Fanuc TP program (LS listing): _set_rack_slot.ls

/PROG  _SET_RACK_SLOT
/ATTR
OWNER		= MNEDITOR;
COMMENT		= "";
PROG_SIZE	= 6875;
CREATE		= DATE 26-07-16  TIME 09:15:24;
MODIFIED	= DATE 26-07-17  TIME 00:46:46;
FILE_NAME	= ;
VERSION		= 0;
LINE_COUNT	= 333;
MEMORY_SIZE	= 7591;
PROTECT		= READ_WRITE;
TCD:  STACK_SIZE	= 0,
      TASK_PRIORITY	= 50,
      TIME_SLICE	= 0,
      BUSY_LAMP_OFF	= 0,
      ABORT_REQUEST	= 0,
      PAUSE_REQUEST	= 0;
DEFAULT_GROUP	= 1,*,*,*,*;
CONTROL_CODE	= 00000000 00000000;
LOCAL_REGISTERS	= 0,0,0;
/APPL

AUTO_SINGULARITY_HEADER;
  ENABLE_SINGULARITY_AVOIDANCE   : TRUE;
/MN
   1:  !*******SET RACK PKPL SLOT******* ;
   2:  LBL[100] ;
   3:  F[21:OFF:Rack Slot-Set]=(OFF) ;
   4:  !**Jump for Rack to PKPL at ;
   5:  SELECT R[20:*RackNum]=1,JMP LBL[210] ;
   6:         =2,JMP LBL[220] ;
   7:         =3,JMP LBL[230] ;
   8:         =4,JMP LBL[240] ;
   9:         =5,JMP LBL[250] ;
  10:         =6,JMP LBL[260] ;
  11:  JMP LBL[700] ;
  12:   ;
  13:  !***Rack-1 (Door)**************** ;
  14:  LBL[210] ;
  15:  !Jump for Column ;
  16:  SELECT R[25:*Slot-Colmn]=1,JMP LBL[211] ;
  17:         =2,JMP LBL[212] ;
  18:         =3,JMP LBL[213] ;
  19:         =4,JMP LBL[214] ;
  20:  JMP LBL[700] ;
  21:   ;
  22:  !**Column 1-Chk Row  ;
  23:  LBL[211] ;
  24:  IF (R[26:*Slot-Row]<1 OR R[26:*Slot-Row]>7),JMP LBL[700] ;
  25:  !Set Origin PR ;
  26:  R[27:*RackOrig-PR]=161    ;
  27:  !Set Appr PR/Transit Angle ;
  28:  R[28:*RackAppr-PR]=131    ;
  29:  R[24:*TransitAngle]=(-155)    ;
  30:  JMP LBL[300] ;
  31:   ;
  32:  !**Column 2-Chk Row  ;
  33:  LBL[212] ;
  34:  IF (R[26:*Slot-Row]<>1 AND R[26:*Slot-Row]<>2),JMP LBL[700] ;
  35:  !Set Origin PR ;
  36:  R[27:*RackOrig-PR]=162    ;
  37:  !Set Appr PR/Transit Angle ;
  38:  R[28:*RackAppr-PR]=131    ;
  39:  R[24:*TransitAngle]=(-155)    ;
  40:  JMP LBL[300] ;
  41:   ;
  42:  !**Column 3-Chk Row  ;
  43:  LBL[213] ;
  44:  IF (R[26:*Slot-Row]<>1 AND R[26:*Slot-Row]<>2),JMP LBL[700] ;
  45:  !Set Origin PR ;
  46:  R[27:*RackOrig-PR]=163    ;
  47:  !Set Appr PR/Transit Angle ;
  48:  R[28:*RackAppr-PR]=132    ;
  49:  R[24:*TransitAngle]=155    ;
  50:  JMP LBL[300] ;
  51:   ;
  52:  !**Column 4-Chk Row  ;
  53:  LBL[214] ;
  54:  IF (R[26:*Slot-Row]<1 OR R[26:*Slot-Row]>6),JMP LBL[700] ;
  55:  !Set Origin PR ;
  56:  R[27:*RackOrig-PR]=164    ;
  57:  !Set Appr PR/Transit Angle ;
  58:  R[28:*RackAppr-PR]=132    ;
  59:  R[24:*TransitAngle]=155    ;
  60:  JMP LBL[300] ;
  61:   ;
  62:   ;
  63:  !***Rack-2 (Full)**************** ;
  64:  LBL[220] ;
  65:  !Jump for Column ;
  66:  SELECT R[25:*Slot-Colmn]=1,JMP LBL[221] ;
  67:         =2,JMP LBL[222] ;
  68:         =3,JMP LBL[223] ;
  69:         =4,JMP LBL[224] ;
  70:  JMP LBL[700] ;
  71:   ;
  72:  !**Column 1-Chk Row  ;
  73:  LBL[221] ;
  74:  IF (R[26:*Slot-Row]<1 OR R[26:*Slot-Row]>7),JMP LBL[700] ;
  75:  !Set Origin PR ;
  76:  R[27:*RackOrig-PR]=166    ;
  77:  !Set Appr PR/Transit Angle ;
  78:  R[28:*RackAppr-PR]=133    ;
  79:  R[24:*TransitAngle]=(-95)    ;
  80:  JMP LBL[300] ;
  81:   ;
  82:  !**Column 2-Chk Row  ;
  83:  LBL[222] ;
  84:  IF (R[26:*Slot-Row]<1 OR R[26:*Slot-Row]>7),JMP LBL[700] ;
  85:  !Set Origin PR ;
  86:  R[27:*RackOrig-PR]=167    ;
  87:  !Set Appr PR/Transit Angle ;
  88:  R[28:*RackAppr-PR]=133    ;
  89:  R[24:*TransitAngle]=(-95)    ;
  90:  JMP LBL[300] ;
  91:   ;
  92:  !**Column 3-Chk Row  ;
  93:  LBL[223] ;
  94:  IF (R[26:*Slot-Row]<1 OR R[26:*Slot-Row]>7),JMP LBL[700] ;
  95:  !Set Origin PR ;
  96:  R[27:*RackOrig-PR]=168    ;
  97:  !Set Appr PR/Transit Angle ;
  98:  R[28:*RackAppr-PR]=134    ;
  99:  R[24:*TransitAngle]=(-145)    ;
 100:  JMP LBL[300] ;
 101:   ;
 102:  !**Column 4-Chk Row  ;
 103:  LBL[224] ;
 104:  IF (R[26:*Slot-Row]<1 OR R[26:*Slot-Row]>6),JMP LBL[700] ;
 105:  !Set Origin PR ;
 106:  R[27:*RackOrig-PR]=169    ;
 107:  !Set Appr PR/Transit Angle ;
 108:  R[28:*RackAppr-PR]=134    ;
 109:  R[24:*TransitAngle]=(-145)    ;
 110:  JMP LBL[300] ;
 111:   ;
 112:   ;
 113:  !***Rack-3 (Convs)*************** ;
 114:  LBL[230] ;
 115:  !Jump for Column ;
 116:  SELECT R[25:*Slot-Colmn]=1,JMP LBL[231] ;
 117:         =2,JMP LBL[232] ;
 118:         =3,JMP LBL[233] ;
 119:         =4,JMP LBL[234] ;
 120:  JMP LBL[700] ;
 121:   ;
 122:  !**Column 1-Chk Row  ;
 123:  LBL[231] ;
 124:  IF (R[26:*Slot-Row]<1 OR R[26:*Slot-Row]>4),JMP LBL[700] ;
 125:  !Set Origin PR ;
 126:  R[27:*RackOrig-PR]=171    ;
 127:  !Set Appr PR/Transit Angle ;
 128:  R[28:*RackAppr-PR]=135    ;
 129:  R[24:*TransitAngle]=(-35)    ;
 130:  JMP LBL[300] ;
 131:   ;
 132:  !**Column 2-Chk Row  ;
 133:  LBL[232] ;
 134:  IF (R[26:*Slot-Row]<1 OR R[26:*Slot-Row]>4),JMP LBL[700] ;
 135:  !Set Origin PR ;
 136:  R[27:*RackOrig-PR]=172    ;
 137:  !Set Appr PR/Transit Angle ;
 138:  R[28:*RackAppr-PR]=135    ;
 139:  R[24:*TransitAngle]=(-35)    ;
 140:  JMP LBL[300] ;
 141:   ;
 142:  !**Column 3-Chk Row  ;
 143:  LBL[233] ;
 144:  IF (R[26:*Slot-Row]<1 OR R[26:*Slot-Row]>4),JMP LBL[700] ;
 145:  !Set Origin PR ;
 146:  R[27:*RackOrig-PR]=173    ;
 147:  !Set Appr PR/Transit Angle ;
 148:  R[28:*RackAppr-PR]=136    ;
 149:  R[24:*TransitAngle]=(-85)    ;
 150:  JMP LBL[300] ;
 151:   ;
 152:  !**Column 4-Chk Row  ;
 153:  LBL[234] ;
 154:  IF (R[26:*Slot-Row]<1 OR R[26:*Slot-Row]>4),JMP LBL[700] ;
 155:  !Set Origin PR ;
 156:  R[27:*RackOrig-PR]=174    ;
 157:  !Set Appr PR/Transit Angle ;
 158:  R[28:*RackAppr-PR]=136    ;
 159:  R[24:*TransitAngle]=(-85)    ;
 160:  JMP LBL[300] ;
 161:   ;
 162:   ;
 163:  !***Rack-4 (Hopper)************** ;
 164:  LBL[240] ;
 165:  !Jump for Column ;
 166:  SELECT R[25:*Slot-Colmn]=1,JMP LBL[241] ;
 167:         =2,JMP LBL[242] ;
 168:         =3,JMP LBL[243] ;
 169:         =4,JMP LBL[244] ;
 170:  JMP LBL[700] ;
 171:   ;
 172:  !**Column 1-Chk Row  ;
 173:  LBL[241] ;
 174:  IF (R[26:*Slot-Row]<>1 AND R[26:*Slot-Row]<>6 AND R[26:*Slot-Row]<>7),JMP LBL[700] ;
 175:  !Set Origin PR ;
 176:  R[27:*RackOrig-PR]=176    ;
 177:  !Set Appr PR/Transit Angle ;
 178:  R[28:*RackAppr-PR]=137    ;
 179:  R[24:*TransitAngle]=25    ;
 180:  JMP LBL[300] ;
 181:   ;
 182:  !**Column 2-Chk Row  ;
 183:  LBL[242] ;
 184:  IF (R[26:*Slot-Row]<>1 AND R[26:*Slot-Row]<>6 AND R[26:*Slot-Row]<>7),JMP LBL[700] ;
 185:  !Set Origin PR ;
 186:  R[27:*RackOrig-PR]=177    ;
 187:  !Set Appr PR/Transit Angle ;
 188:  R[28:*RackAppr-PR]=137    ;
 189:  R[24:*TransitAngle]=25    ;
 190:  JMP LBL[300] ;
 191:   ;
 192:  !**Column 3-Chk Row  ;
 193:  LBL[243] ;
 194:  IF (R[26:*Slot-Row]<>1 AND R[26:*Slot-Row]<>6 AND R[26:*Slot-Row]<>7),JMP LBL[700] ;
 195:  !Set Origin PR ;
 196:  R[27:*RackOrig-PR]=178    ;
 197:  !Set Appr PR/Transit Angle ;
 198:  R[28:*RackAppr-PR]=138    ;
 199:  R[24:*TransitAngle]=(-25)    ;
 200:  JMP LBL[300] ;
 201:   ;
 202:  !**Column 4-Chk Row  ;
 203:  LBL[244] ;
 204:  IF (R[26:*Slot-Row]<1 OR R[26:*Slot-Row]>7),JMP LBL[700] ;
 205:  !Set Origin PR ;
 206:  R[27:*RackOrig-PR]=179    ;
 207:  !Set Appr PR/Transit Angle ;
 208:  R[28:*RackAppr-PR]=138    ;
 209:  R[24:*TransitAngle]=(-25)    ;
 210:  JMP LBL[300] ;
 211:   ;
 212:   ;
 213:  !***Rack-5 (Full)**************** ;
 214:  LBL[250] ;
 215:  !Jump for Column ;
 216:  SELECT R[25:*Slot-Colmn]=1,JMP LBL[251] ;
 217:         =2,JMP LBL[252] ;
 218:         =3,JMP LBL[253] ;
 219:         =4,JMP LBL[254] ;
 220:  JMP LBL[700] ;
 221:   ;
 222:  !**Column 1-Chk Row  ;
 223:  LBL[251] ;
 224:  IF (R[26:*Slot-Row]<1 OR R[26:*Slot-Row]>7),JMP LBL[700] ;
 225:  !Set Origin PR ;
 226:  R[27:*RackOrig-PR]=181    ;
 227:  !Set Appr PR/Transit Angle ;
 228:  R[28:*RackAppr-PR]=139    ;
 229:  R[24:*TransitAngle]=85    ;
 230:  JMP LBL[300] ;
 231:   ;
 232:  !**Column 2-Chk Row  ;
 233:  LBL[252] ;
 234:  IF (R[26:*Slot-Row]<1 OR R[26:*Slot-Row]>7),JMP LBL[700] ;
 235:  !Set Origin PR ;
 236:  R[27:*RackOrig-PR]=182    ;
 237:  !Set Appr PR/Transit Angle ;
 238:  R[28:*RackAppr-PR]=139    ;
 239:  R[24:*TransitAngle]=85    ;
 240:  JMP LBL[300] ;
 241:   ;
 242:  !**Column 3-Chk Row  ;
 243:  LBL[253] ;
 244:  IF (R[26:*Slot-Row]<1 OR R[26:*Slot-Row]>7),JMP LBL[700] ;
 245:  !Set Origin PR ;
 246:  R[27:*RackOrig-PR]=183    ;
 247:  !Set Appr PR/Transit Angle ;
 248:  R[28:*RackAppr-PR]=140    ;
 249:  R[24:*TransitAngle]=35    ;
 250:  JMP LBL[300] ;
 251:   ;
 252:  !**Column 4-Chk Row  ;
 253:  LBL[254] ;
 254:  IF (R[26:*Slot-Row]<1 OR R[26:*Slot-Row]>7),JMP LBL[700] ;
 255:  !Set Origin PR ;
 256:  R[27:*RackOrig-PR]=184    ;
 257:  !Set Appr PR/Transit Angle ;
 258:  R[28:*RackAppr-PR]=140    ;
 259:  R[24:*TransitAngle]=35    ;
 260:  JMP LBL[300] ;
 261:   ;
 262:   ;
 263:  !***Rack-6 (Full)**************** ;
 264:  LBL[260] ;
 265:  !Jump for Column ;
 266:  SELECT R[25:*Slot-Colmn]=1,JMP LBL[261] ;
 267:         =2,JMP LBL[262] ;
 268:         =3,JMP LBL[263] ;
 269:         =4,JMP LBL[264] ;
 270:  JMP LBL[700] ;
 271:   ;
 272:  !**Column 1-Chk Row  ;
 273:  LBL[261] ;
 274:  IF (R[26:*Slot-Row]<1 OR R[26:*Slot-Row]>6),JMP LBL[700] ;
 275:  !Set Origin PR ;
 276:  R[27:*RackOrig-PR]=186    ;
 277:  !Set Appr PR/Transit Angle ;
 278:  R[28:*RackAppr-PR]=141    ;
 279:  R[24:*TransitAngle]=145    ;
 280:  JMP LBL[300] ;
 281:   ;
 282:  !**Column 2-Chk Row  ;
 283:  LBL[262] ;
 284:  IF (R[26:*Slot-Row]<1 OR R[26:*Slot-Row]>6),JMP LBL[700] ;
 285:  !Set Origin PR ;
 286:  R[27:*RackOrig-PR]=187    ;
 287:  !Set Appr PR/Transit Angle ;
 288:  R[28:*RackAppr-PR]=141    ;
 289:  R[24:*TransitAngle]=145    ;
 290:  JMP LBL[300] ;
 291:   ;
 292:  !**Column 3-Chk Row  ;
 293:  LBL[263] ;
 294:  IF (R[26:*Slot-Row]<1 OR R[26:*Slot-Row]>7),JMP LBL[700] ;
 295:  !Set Origin PR ;
 296:  R[27:*RackOrig-PR]=188    ;
 297:  !Set Appr PR/Transit Angle ;
 298:  R[28:*RackAppr-PR]=142    ;
 299:  R[24:*TransitAngle]=95    ;
 300:  JMP LBL[300] ;
 301:   ;
 302:  !**Column 4-Chk Row  ;
 303:  LBL[264] ;
 304:  IF (R[26:*Slot-Row]<1 OR R[26:*Slot-Row]>7),JMP LBL[700] ;
 305:  !Set Origin PR ;
 306:  R[27:*RackOrig-PR]=189    ;
 307:  !Set Appr PR/Transit Angle ;
 308:  R[28:*RackAppr-PR]=142    ;
 309:  R[24:*TransitAngle]=95    ;
 310:  JMP LBL[300] ;
 311:  !******************************** ;
 312:   ;
 313:   ;
 314:  !**********SET SLOT NUM********** ;
 315:  LBL[300] ;
 316:  R[91:*tempX]=((R[20:*RackNum]-1)*28) ;
 317:  R[92:*tempY]=((R[25:*Slot-Colmn]-1)*7) ;
 318:  R[21:*SlotNum]=R[91:*tempX]+R[92:*tempY]+R[26:*Slot-Row]    ;
 319:  JMP LBL[900] ;
 320:   ;
 321:   ;
 322:  !*********SET SLOT ERROR********* ;
 323:  LBL[700] ;
 324:  F[21:OFF:Rack Slot-Set]=(OFF) ;
 325:  JMP LBL[999] ;
 326:   ;
 327:  !*********RACK SLOT SET********** ;
 328:  LBL[900] ;
 329:  F[21:OFF:Rack Slot-Set]=(ON) ;
 330:  JMP LBL[999] ;
 331:   ;
 332:   ;
 333:  LBL[999] ;
/POS
/END
